RoboDK station: AccelerationCalculation.rdk

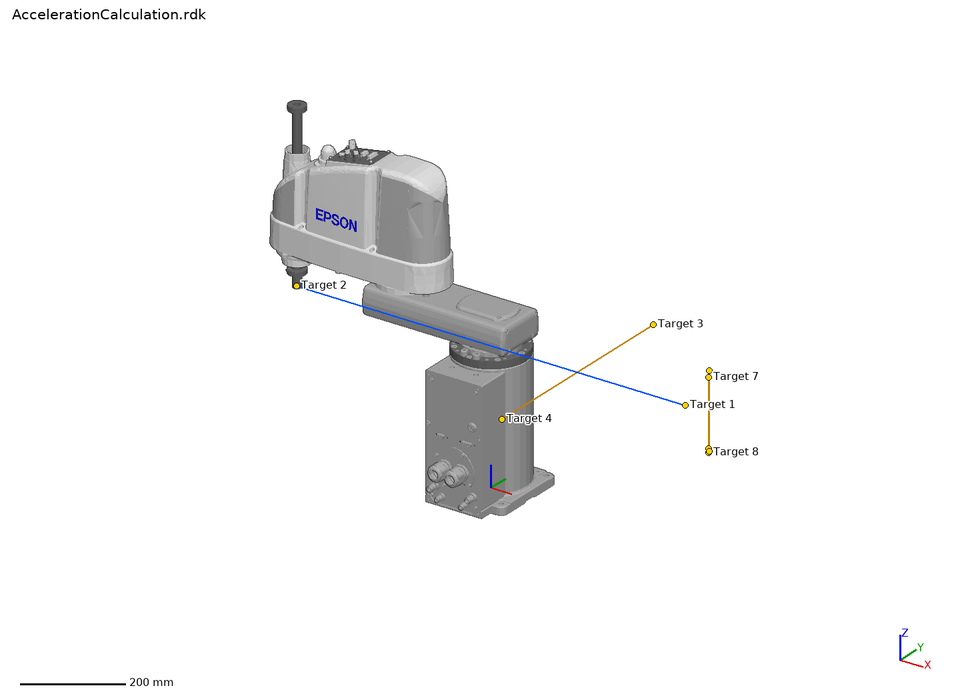
[picture v0: the station drawn from its stored meshes, robots at their saved joint values, targets as dots, program paths as lines]
Station AccelerationCalculation (saved by RoboDK 5.9.6). Poses are relative to the parent item; angles as X-Y-Z fixed-axis rotations.
  - frame Epson_G6_451s Base at (0, 0, 0) mm
    - robot Epson_G6_451s: 4 axes
        modified DH rows (alpha deg, a mm, theta deg, d mm): 0, 0, 0, 0; 0, 200, 0, 0; 0, 250, 0, -180 linear; 180, 0, 0, 0
        joint limits [-62, -142, -180, -360] to [242, 142, 0, 360]; home [0, 0, 0, 0]; saved at [180, 0, 0, 0]
    - target Target 1 (Cartesian target) at (450, 0, 300) mm, rotated rx 180 ry 0 rz 0 deg; joints [0, 0, 0, 0] of Epson_G6_451s
    - target Target 2 (Cartesian target) at (-450, 0, 300) mm, rotated rx 180 ry 0 rz 180 deg; joints [180, 0, 0, 0] of Epson_G6_451s
    - target Target 3 (Cartesian target) at (200, 250, 300) mm, rotated rx 180 ry 0 rz 90 deg; joints [0, 90, 0, 0] of Epson_G6_451s
    - target Target 4 (Cartesian target) at (200, -250, 300) mm, rotated rx 180 ry 0 rz -90 deg; joints [0, -90, 0, 0] of Epson_G6_451s
    - target Target 5 (Cartesian target) at (200, 250, 300) mm, rotated rx 180 ry 0 rz 90 deg; joints [0, 90, 0, 0] of Epson_G6_451s
    - target Target 6 (Cartesian target) at (450, 0, 300) mm, rotated rx 180 ry 0 rz 0 deg; joints [0, 0, 0, 0] of Epson_G6_451s
    - target Target 7 (Cartesian target) at (416.68, 124.7, 300) mm, rotated rx 180 ry 0 rz 29.92 deg; joints [0, 29.92, 0, 0] of Epson_G6_451s
    - target Target 8 (Cartesian target) at (416.68, 124.7, 141) mm, rotated rx 180 ry 0 rz 29.92 deg; joints [0, 29.92, -159, 0] of Epson_G6_451s
    - target Target 9 (Cartesian target) at (416.68, 124.7, 150) mm, rotated rx 180 ry 0 rz 29.92 deg; joints [0, 29.92, -150, 0] of Epson_G6_451s
    - target Target 10 (Cartesian target) at (450, 0, 300) mm, rotated rx 180 ry 0 rz 0 deg; joints [0, 0, 0, 0] of Epson_G6_451s
    - target Target 11 (Cartesian target) at (-450, 0, 300) mm, rotated rx 180 ry 0 rz 180 deg; joints [180, 0, 0, 0] of Epson_G6_451s
    - target Target 12 (Cartesian target) at (400.78, 148.95, 130) mm, rotated rx 180 ry 0 rz 36.57 deg; joints [0, 36.57, -170, 0] of Epson_G6_451s
    - target Target 13 (Cartesian target) at (400.78, 148.95, 300) mm, rotated rx 180 ry 0 rz 36.57 deg; joints [0, 36.57, 0, 0] of Epson_G6_451s
    - target Target 14 (Cartesian target) at (450, 0, 300) mm, rotated rx 180 ry 0 rz -10 deg; joints [0, 0, 0, -350] of Epson_G6_451s
    - target Target 15 (Cartesian target) at (450, 0, 300) mm, rotated rx 180 ry 0 rz 10 deg; joints [0, 0, 0, 350] of Epson_G6_451s
  - program Joint1 (4 instructions, listed below)
  - Python program GetJointData (listed below)
  - program Joint2 (3 instructions, listed below)
  - program Joint3_Power (61 instructions, listed below)
  - program Joint1_Power (51 instructions, listed below)
  - program Joint2_Power (70 instructions, listed below)
  - program Joint3 (4 instructions, listed below)
  - program Prog6 (5 instructions, listed below)
  - Python program SpeedOutput (listed below)
  - Python program FullOutput (listed below)
  - Python program FullOutputCSVJointMove (listed below)
  - Python program FullOutputCSVLinearMove (listed below)
  - Python program Prog9 (listed below)
  - program Prog14 (61 instructions, listed below)
  - program Joint4 (3 instructions, listed below)
  - program Joint4_Power (60 instructions, listed below)
  - program Prog17 (10 instructions, listed below)
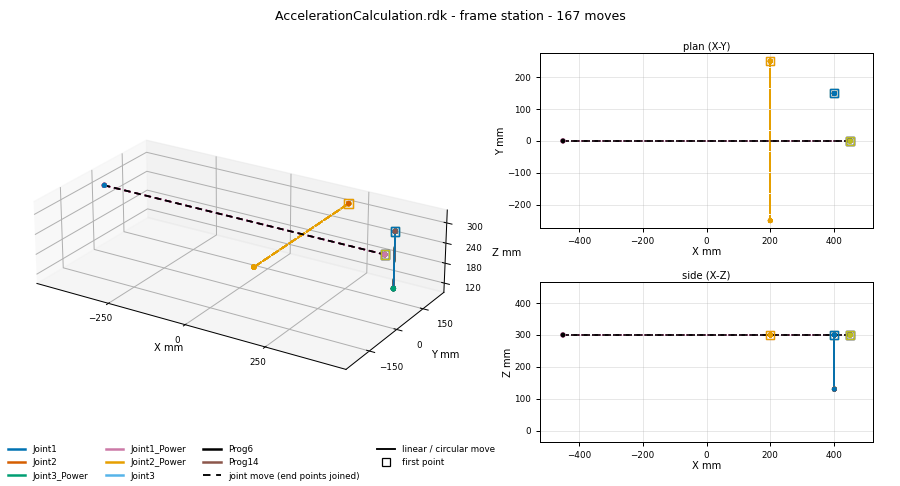
[picture p0: tool path of AccelerationCalculation.rdk in frame station, 167 of 167 moves have a stored position in this frame; points joined in program order, loops and branches not executed]

--- program Joint1 (robot Epson_G6_451s) ---
  Set Ref.: Epson_G6_451s Base
  Set speed (42.0 deg/s)
  MoveJ (Target 1)
  MoveJ (Target 2)

--- Python program GetJointData ---
from robodk import robolink, robomath
import matplotlib.pyplot as plt
from robodk.robolink import *
from robodk.robomath import *
import csv

# Connect to RoboDK
RDK = Robolink()


# Select your program by name
program = RDK.Item('Joint1', robolink.ITEM_TYPE_PROGRAM)  # Change name as needed

# Run the program (optional — comment out if already simulated)
program.RunProgram()

# Retrieve joint data
data_all = program.InstructionListJoints(mm_step=1, deg_step=1, flags=3)
data_all = data_all[1:]

joint_data = data_all[0]
print(joint_data)

# Output file path (can be absolute or relative)
csv_file = 'C:/Users/kytho/Desktop/robot_data.csv'

if program.Valid():
    # Write to CSV

    # Add header row (titles) and append a cumulative Time_Total column
    header = [
        'J1_Position', 'J2_Position', 'J3_Position', 'J4_Position', 'Error',
        'MM_Step', 'Deg_step', 'Move_ID', 'Time', 'Time_Total', 'X', 'Y', 'Z',
        'J1_Velocity', 'J2_Velocity', 'J3_Velocity', 'J4_Velocity',
        'J1_Acceleration', 'J2_Acceleration', 'J3_Acceleration', 'J4_Acceleration'
    ]

    with open(csv_file, "w", newline="") as file:
        writer = csv.writer(file)
        # write header first (move all data one row down)
        writer.writerow(header)

        # compute cumulative Time_Total (Time is expected at index 8)
        time_total = 0.0
        for row in joint_data:
            # keep the original data unchanged; append Time_Total after Time
            new_row = list(row)
            try:
                # read time delta from column index 8
                t_delta = float(row[8])
            except Exception:
                # if parsing fails, treat delta as 0.0
                t_delta = 0.0
            time_total += t_delta
            # insert cumulative time after the existing Time column
            new_row.insert(9, time_total)
            writer.writerow(new_row)

    print("Joint data successfully written to 'robot_data.csv'")
    print("Total Time:",time_total)
else:
    print("No valid program selected.")

--- program Joint2 (robot Epson_G6_451s) ---
  Set Ref.: Epson_G6_451s Base
  MoveJ (Target 5)
  MoveJ (Target 4)

--- program Joint3_Power (robot Epson_G6_451s) ---
  Set Ref.: Epson_G6_451s Base
  Set speed (1182.2 mm/s)
  MoveJ (Target 13)
  MoveL (Target 13)
  MoveL (Target 12)
  Pause 1.0 s
  MoveL (Target 13)
  Pause 1.0 s
  Set speed (1070.0 mm/s)
  MoveL (Target 13)
  MoveL (Target 12)
  Pause 1.0 s
  MoveL (Target 13)
  Pause 1.0 s
  Set speed (953.1 mm/s)
  MoveL (Target 13)
  MoveL (Target 12)
  Pause 1.0 s
  MoveL (Target 13)
  Pause 1.0 s
  Set speed (828.6 mm/s)
  MoveL (Target 13)
  MoveL (Target 12)
  Pause 1.0 s
  MoveL (Target 13)
  Pause 1.0 s
  Set speed (716.0 mm/s)
  MoveL (Target 13)
  MoveL (Target 12)
  Pause 1.0 s
  MoveL (Target 13)
  Pause 1.0 s
  Set speed (595.8 mm/s)
  MoveL (Target 13)
  MoveL (Target 12)
  Pause 1.0 s
  MoveL (Target 13)
  Pause 1.0 s
  Set speed (477.4 mm/s)
  MoveL (Target 13)
  MoveL (Target 12)
  Pause 1.0 s
  MoveL (Target 13)
  Pause 1.0 s
  Set speed (358.1 mm/s)
  MoveL (Target 13)
  MoveL (Target 12)
  Pause 1.0 s
  MoveL (Target 13)
  Pause 1.0 s
  Set speed (238.7 mm/s)
  MoveL (Target 13)
  MoveL (Target 12)
  Pause 1.0 s
  MoveL (Target 13)
  Pause 1.0 s
  Set speed (119.3 mm/s)
  MoveL (Target 13)
  MoveL (Target 12)
  Pause 1.0 s
  MoveL (Target 13)

--- program Joint1_Power (robot Epson_G6_451s) ---
  Set Ref.: Epson_G6_451s Base
  Set speed (420.0 deg/s)
  MoveJ (Target 10)
  MoveJ (Target 11)
  MoveJ (Target 10)
  Pause 1.0 s
  Set speed (378.0 deg/s)
  MoveJ (Target 10)
  MoveJ (Target 11)
  MoveJ (Target 10)
  Pause 1.0 s
  Set speed (336.0 deg/s)
  MoveJ (Target 10)
  MoveJ (Target 11)
  MoveJ (Target 10)
  Pause 1.0 s
  Set speed (294.0 deg/s)
  MoveJ (Target 10)
  MoveJ (Target 11)
  MoveJ (Target 10)
  Pause 1.0 s
  Set speed (251.0 deg/s)
  MoveJ (Target 10)
  MoveJ (Target 11)
  MoveJ (Target 10)
  Pause 1.0 s
  Set speed (210.0 deg/s)
  MoveJ (Target 10)
  MoveJ (Target 11)
  MoveJ (Target 10)
  Pause 1.0 s
  Set speed (168.0 deg/s)
  MoveJ (Target 10)
  MoveJ (Target 11)
  MoveJ (Target 10)
  Pause 1.0 s
  Set speed (126.0 deg/s)
  MoveJ (Target 10)
  MoveJ (Target 11)
  MoveJ (Target 10)
  Pause 1.0 s
  Set speed (84.0 deg/s)
  MoveJ (Target 10)
  MoveJ (Target 11)
  MoveJ (Target 10)
  Pause 1.0 s
  Set speed (42.0 deg/s)
  MoveJ (Target 10)
  MoveJ (Target 11)
  MoveJ (Target 10)
  Pause 1.0 s

--- program Joint2_Power (robot Epson_G6_451s) ---
  Set speed (720.0 deg/s)
  Set Ref.: Epson_G6_451s Base
  MoveJ (Target 5)
  MoveJ (Target 4)
  Pause 1.0 s
  MoveJ (Target 5)
  Pause 1.0 s
  Set speed (648.0 deg/s)
  Set Ref.: Epson_G6_451s Base
  MoveJ (Target 5)
  MoveJ (Target 4)
  Pause 1.0 s
  MoveJ (Target 5)
  Pause 1.0 s
  Set speed (576.0 deg/s)
  Set Ref.: Epson_G6_451s Base
  MoveJ (Target 5)
  MoveJ (Target 4)
  Pause 1.0 s
  MoveJ (Target 5)
  Pause 1.0 s
  Set speed (504.0 deg/s)
  Set Ref.: Epson_G6_451s Base
  MoveJ (Target 5)
  MoveJ (Target 4)
  Pause 1.0 s
  MoveJ (Target 5)
  Pause 1.0 s
  Set speed (432.0 deg/s)
  Set Ref.: Epson_G6_451s Base
  MoveJ (Target 5)
  MoveJ (Target 4)
  Pause 1.0 s
  MoveJ (Target 5)
  Pause 1.0 s
  Set speed (360.0 deg/s)
  Set Ref.: Epson_G6_451s Base
  MoveJ (Target 5)
  MoveJ (Target 4)
  Pause 1.0 s
  MoveJ (Target 5)
  Pause 1.0 s
  Set speed (288.0 deg/s)
  Set Ref.: Epson_G6_451s Base
  MoveJ (Target 5)
  MoveJ (Target 4)
  Pause 1.0 s
  MoveJ (Target 5)
  Pause 1.0 s
  Set speed (216.0 deg/s)
  Set Ref.: Epson_G6_451s Base
  MoveJ (Target 5)
  MoveJ (Target 4)
  Pause 1.0 s
  MoveJ (Target 5)
  Pause 1.0 s
  Set speed (144.0 deg/s)
  Set Ref.: Epson_G6_451s Base
  MoveJ (Target 5)
  MoveJ (Target 4)
  Pause 1.0 s
  MoveJ (Target 5)
  Pause 1.0 s
  Set speed (72.0 deg/s)
  Set Ref.: Epson_G6_451s Base
  MoveJ (Target 5)
  MoveJ (Target 4)
  Pause 1.0 s
  MoveJ (Target 5)
  Pause 1.0 s

--- program Joint3 (robot Epson_G6_451s) ---
  Set Ref.: Epson_G6_451s Base
  Set speed (500.0 mm/s)
  MoveL (Target 13)
  MoveL (Target 12)

--- program Prog6 (robot Epson_G6_451s) ---
  Set Ref.: Epson_G6_451s Base
  Set speed (41.0 deg/s)
  MoveJ (Target 10)
  MoveJ (Target 11)
  MoveJ (Target 10)

--- Python program SpeedOutput ---
# This example shows how to quickly calculate the cycle time of a program
# as a function of the linear and joint speeds
#
# Important notes and tips for accurate cycle time calculation:
# https://robodk.com/doc/en/General.html#CycleTime

# Start the RoboDK API
from robodk.robolink import *  # RoboDK API

RDK = Robolink()

# Ask the user to select a program
program = RDK.ItemUserPick('Joint2', ITEM_TYPE_PROGRAM)

# Retrieve the robot linked to the selected program
robot = program.getLink(ITEM_TYPE_ROBOT)

for speed_joints in range(20, 601, 10):
    # Set the robot speed
    robot.setAcceleration(3516.67)
    robot.setSpeed(500, speed_joints)
    # Update the program and retrieve updated information:
    # https://robodk.com/doc/en/PythonAPI/robodk.html#robodk.robolink.Item.Update
    result = program.Update()
    instructions, time, travel, ok, error = result

    # Print the information
    print("Speed", speed_joints)
    print(time)

--- Python program FullOutput ---
# This example shows how to quickly calculate the cycle time of a program
# as a function of the linear and joint speeds
#
# Important notes and tips for accurate cycle time calculation:
# https://robodk.com/doc/en/General.html#CycleTime

# Start the RoboDK API
from robodk.robolink import *  # RoboDK API

RDK = Robolink()

# Ask the user to select a program
program = RDK.ItemUserPick('Joint2', ITEM_TYPE_PROGRAM)

# Retrieve the robot linked to the selected program
robot = program.getLink(ITEM_TYPE_ROBOT)

for speed_joints in range(20, 601, 10):
    # Set the robot speed
    robot.setAccelerationJoints(3516.67)
    robot.setSpeed(500, speed_joints)
    # Update the program and retrieve updated information:
    # https://robodk.com/doc/en/PythonAPI/robodk.html#robodk.robolink.Item.Update
    result = program.Update()
    instructions, time, travel, ok, error = result

    # Print the information
    print("Speed", speed_joints)
    print(time)

for accel_joints in range(100, 4001, 100):
    # Set the robot speed
    robot.setAccelerationJoints(accel_joints)
    robot.setSpeed(500, 520)
    # Update the program and retrieve updated information:
    # https://robodk.com/doc/en/PythonAPI/robodk.html#robodk.robolink.Item.Update
    result = program.Update()
    instructions, time2, travel, ok, error = result

    # Print the information
    print("Acceleration:", accel_joints)
    print(time2)

--- Python program FullOutputCSVJointMove ---
# This example calculates program cycle time as a function of
# joint speed and joint acceleration and writes results to CSV

from robodk.robolink import *  # RoboDK API
import csv
import os

RDK = Robolink()

# Select program
program = RDK.ItemUserPick('Select a program', ITEM_TYPE_PROGRAM)
if not program.Valid():
    raise Exception("No program selected.")

# Get linked robot
robot = program.getLink(ITEM_TYPE_ROBOT)
if not robot.Valid():
    raise Exception("No robot linked to program.")

results = []

# -----------------------------
# SPEED SWEEP
# -----------------------------
for speed_joints in range(20, 3400, 50):

    robot.setAccelerationJoints(1645.795918)
    robot.setSpeed(500, speed_joints)

    result = program.Update()
    instructions, time_val, travel, ok, error = result

    print("Speed:", speed_joints)
    print("Cycle Time:", time_val)

    results.append([speed_joints, time_val, "", ""])

# -----------------------------
# ACCELERATION SWEEP
# -----------------------------
for accel_joints in range(100, 15100, 100):

    robot.setAccelerationJoints(accel_joints)
    robot.setSpeed(1, 420)

    result = program.Update()
    instructions, time_val, travel, ok, error = result

    print("Acceleration:", accel_joints)
    print("Cycle Time:", time_val)

    results.append(["", "", accel_joints, time_val])

# -----------------------------
# WRITE CSV
# -----------------------------
filename = "robodk_cycle_time_results.csv"

with open(filename, mode='w', newline='') as file:
    writer = csv.writer(file)
    writer.writerow(["joint_speed", "cycle_time", "joint_accel", "cycle_time"])
    writer.writerows(results)

print("\nResults saved to:", os.path.abspath(filename))

--- Python program FullOutputCSVLinearMove ---
# This example calculates program cycle time as a function of
# joint speed and joint acceleration and writes results to CSV

from robodk.robolink import *  # RoboDK API
import csv
import os

RDK = Robolink()

# Select program
program = RDK.ItemUserPick('Select a program', ITEM_TYPE_PROGRAM)
if not program.Valid():
    raise Exception("No program selected.")

# Get linked robot
robot = program.getLink(ITEM_TYPE_ROBOT)
if not robot.Valid():
    raise Exception("No robot linked to program.")

results = []

# -----------------------------
# SPEED SWEEP
# -----------------------------
for speed_joints in range(20, 2001, 20):

    robot.setAcceleration(10100.434747)
    robot.setSpeed(speed_joints, 480)

    result = program.Update()
    instructions, time_val, travel, ok, error = result

    print("Speed:", speed_joints)
    print("Cycle Time:", time_val)

    results.append([speed_joints, time_val, "", ""])

# -----------------------------
# ACCELERATION SWEEP
# -----------------------------
for accel_joints in range(100, 50000, 200):

    robot.setAcceleration(accel_joints)
    robot.setSpeed(1180, 480.037)

    result = program.Update()
    instructions, time_val, travel, ok, error = result

    print("Acceleration:", accel_joints)
    print("Cycle Time:", time_val)

    results.append(["", "", accel_joints, time_val])

# -----------------------------
# WRITE CSV
# -----------------------------
filename = "robodk_cycle_time_results.csv"

with open(filename, mode='w', newline='') as file:
    writer = csv.writer(file)
    writer.writerow(["joint_speed", "cycle_time", "joint_accel", "cycle_time"])
    writer.writerows(results)

print("\nResults saved to:", os.path.abspath(filename))

--- Python program Prog9 ---
from robodk.robolink import Robolink, ITEM_TYPE_PROGRAM
import csv
import re
import statistics
from collections import defaultdict

PROGRAM_NAME = "Joint1_Power"
OUT_CSV = r"C:/Users/kytho/Desktop/robot_data_with_pauses.csv"

def pick_pause_dt(joint_rows, dt_index=8):
    """Use median dt from motion samples for pause sampling."""
    dts = []
    for r in joint_rows:
        try:
            dt = float(r[dt_index])
            if dt > 0:
                dts.append(dt)
        except:
            pass
    return statistics.median(dts) if dts else 0.01

def get_events_from_program_tree(program):
    """
    Build ordered events by reading instruction nodes from the RoboDK tree.
    Requires program.ShowInstructions(True).
    """
    program.ShowInstructions(True)  # key workaround: expose instruction nodes in tree

    children = program.Childs()  # returns items in program order (tree order)
    events = []

    # Matches: "Pause 1.0 s" / "Pause 1s" / "Pause 0.5 s"
    pause_re = re.compile(r"^\s*Pause\s*([0-9]*\.?[0-9]+)\s*s?\s*$", re.IGNORECASE)

    for it in children:
        name = it.Name().strip()

        m = pause_re.match(name)
        if m:
            events.append(("PAUSE", float(m.group(1))))
            continue

        n = name.lower()
        if n.startswith("movej") or n.startswith("movel") or n.startswith("movec"):
            events.append(("MOVE", None))
            continue

        # Ignore "Set speed", messages, etc. (add here if you want them handled)

    return events

def main():
    RDK = Robolink()

    program = RDK.Item(PROGRAM_NAME, ITEM_TYPE_PROGRAM)
    if not program.Valid():
        raise Exception(f"Program not found: {PROGRAM_NAME}")

    # --- motion samples (movement only) ---
    data_all = program.InstructionListJoints(mm_step=1, deg_step=1, flags=3)
    data_all = data_all[1:]  # skip header block if present
    joint_rows = data_all[0]
    if not joint_rows:
        raise Exception("No joint data returned by InstructionListJoints().")

    IDX_MOVE_ID = 7
    IDX_DT = 8

    # Group rows by Move_ID in appearance order
    rows_by_move = defaultdict(list)
    move_ids_in_order = []
    seen = set()
    for row in joint_rows:
        mid = row[IDX_MOVE_ID]
        rows_by_move[mid].append(row)
        if mid not in seen:
            seen.add(mid)
            move_ids_in_order.append(mid)

    # --- parse events from program tree (includes Pause items) ---
    events = get_events_from_program_tree(program)

    move_events = sum(1 for e in events if e[0] == "MOVE")
    pause_events = sum(1 for e in events if e[0] == "PAUSE")
    print("MOVE events found:", move_events)
    print("PAUSE events found:", pause_events)

    if pause_events == 0:
        print("WARNING: No pauses detected from program tree items. Check that pause items exist and are named like 'Pause 1.0 s'.")
    if move_events == 0:
        print("WARNING: No MOVE events detected from program tree items. Check that the program contains MoveJ/MoveL instructions.")

    pause_dt = pick_pause_dt(joint_rows, dt_index=IDX_DT)

    # Output header (same as yours)
    header = [
        "J1_Position", "J2_Position", "J3_Position", "J4_Position", "Error",
        "MM_Step", "Deg_step", "Move_ID", "Time", "Time_Total", "X", "Y", "Z",
        "J1_Velocity", "J2_Velocity", "J3_Velocity", "J4_Velocity",
        "J1_Acceleration", "J2_Acceleration", "J3_Acceleration", "J4_Acceleration"
    ]

    time_total = 0.0
    move_ptr = 0
    last_written = None

    with open(OUT_CSV, "w", newline="") as f:
        w = csv.writer(f)
        w.writerow(header)

        for ev_type, ev_val in events:
            if ev_type == "MOVE":
                if move_ptr >= len(move_ids_in_order):
                    continue

                mid = move_ids_in_order[move_ptr]
                move_ptr += 1

                for row in rows_by_move[mid]:
                    new_row = list(row)
                    try:
                        dt = float(row[IDX_DT])
                    except:
                        dt = 0.0

                    time_total += dt
                    new_row.insert(9, time_total)  # Time_Total after Time column
                    w.writerow(new_row)
                    last_written = new_row

            elif ev_type == "PAUSE":
                pause_s = float(ev_val)
                if last_written is None:
                    continue

                remaining = pause_s
                while remaining > 1e-12:
                    dt = pause_dt if remaining > pause_dt else remaining
                    remaining -= dt

                    pause_row = list(last_written)

                    # "Time" is at index 8, "Time_Total" at index 9 (because we inserted it)
                    pause_row[8] = dt

                    # Zero velocities (cols 13..16) and accelerations (17..20)
                    for i in range(13, 17):
                        pause_row[i] = 0.0
                    for i in range(17, 21):
                        pause_row[i] = 0.0

                    time_total += dt
                    pause_row[9] = time_total
                    w.writerow(pause_row)
                    last_written = pause_row

        # Append any leftover motion blocks if events had fewer MOVE entries than motion blocks
        while move_ptr < len(move_ids_in_order):
            mid = move_ids_in_order[move_ptr]
            move_ptr += 1
            for row in rows_by_move[mid]:
                new_row = list(row)
                try:
                    dt = float(row[IDX_DT])
                except:
                    dt = 0.0
                time_total += dt
                new_row.insert(9, time_total)
                w.writerow(new_row)

    print("Wrote:", OUT_CSV)
    print("Total time (motion + inserted pauses):", time_total)

if __name__ == "__main__":
    main()

--- program Prog14 (robot Epson_G6_451s) ---
  Set Ref.: Epson_G6_451s Base
  Set speed (1100.0 mm/s)
  MoveJ (Target 13)
  MoveL (Target 12)
  Pause 1.0 s
  MoveL (Target 13)
  Pause 1.0 s
  Set speed (990.0 mm/s)
  MoveJ (Target 13)
  MoveL (Target 12)
  Pause 1.0 s
  MoveL (Target 13)
  Pause 1.0 s
  Set speed (880.0 mm/s)
  MoveJ (Target 13)
  MoveL (Target 12)
  Pause 1.0 s
  MoveL (Target 13)
  Pause 1.0 s
  Set speed (770.0 mm/s)
  MoveJ (Target 13)
  MoveL (Target 12)
  Pause 1.0 s
  MoveL (Target 13)
  Pause 1.0 s
  Set speed (660.0 mm/s)
  MoveJ (Target 13)
  MoveL (Target 12)
  Pause 1.0 s
  MoveL (Target 13)
  Pause 1.0 s
  Set speed (550.0 mm/s)
  MoveJ (Target 13)
  MoveL (Target 12)
  Pause 1.0 s
  MoveL (Target 13)
  Pause 1.0 s
  Set speed (440.0 mm/s)
  MoveJ (Target 13)
  MoveL (Target 12)
  Pause 1.0 s
  MoveL (Target 13)
  Pause 1.0 s
  Set speed (330.0 mm/s)
  MoveJ (Target 13)
  MoveL (Target 12)
  Pause 1.0 s
  MoveL (Target 13)
  Pause 1.0 s
  Set speed (220.0 mm/s)
  MoveJ (Target 13)
  MoveL (Target 12)
  Pause 1.0 s
  MoveL (Target 13)
  Pause 1.0 s
  Set speed (110.0 mm/s)
  MoveJ (Target 13)
  MoveL (Target 12)
  Pause 1.0 s
  MoveL (Target 13)
  Pause 1.0 s

--- program Joint4 (robot Epson_G6_451s) ---
  Set Ref.: Epson_G6_451s Base
  MoveJ (Target 14)
  MoveJ (Target 15)

--- program Joint4_Power (robot Epson_G6_451s) ---
  Set Ref.: Epson_G6_451s Base
  Set speed (2400.0 deg/s)
  MoveJ (Target 14)
  MoveJ (Target 15)
  Pause 1.0 s
  MoveJ (Target 14)
  Pause 1.0 s
  Set speed (2160.0 deg/s)
  MoveJ (Target 14)
  MoveJ (Target 15)
  Pause 1.0 s
  MoveJ (Target 14)
  Pause 1.0 s
  Set speed (1920.0 deg/s)
  MoveJ (Target 14)
  MoveJ (Target 15)
  Pause 1.0 s
  MoveJ (Target 14)
  Pause 1.0 s
  Set speed (1680.0 deg/s)
  MoveJ (Target 15)
  Pause 1.0 s
  MoveJ (Target 14)
  Pause 1.0 s
  Set speed (1440.7 deg/s)
  MoveJ (Target 14)
  MoveJ (Target 15)
  Pause 1.0 s
  MoveJ (Target 14)
  Pause 1.0 s
  Set speed (1200.0 deg/s)
  MoveJ (Target 14)
  MoveJ (Target 15)
  Pause 1.0 s
  MoveJ (Target 14)
  Pause 1.0 s
  Set speed (960.0 deg/s)
  MoveJ (Target 14)
  MoveJ (Target 15)
  Pause 1.0 s
  MoveJ (Target 14)
  Pause 1.0 s
  Set speed (720.0 deg/s)
  MoveJ (Target 14)
  MoveJ (Target 15)
  Pause 1.0 s
  MoveJ (Target 14)
  Pause 1.0 s
  Set speed (480.0 deg/s)
  MoveJ (Target 14)
  MoveJ (Target 15)
  Pause 1.0 s
  MoveJ (Target 14)
  Pause 1.0 s
  Set speed (240.0 deg/s)
  MoveJ (Target 14)
  MoveJ (Target 15)
  Pause 1.0 s
  MoveJ (Target 14)
  Pause 1.0 s

--- program Prog17 (robot Epson_G6_451s) ---
  Set Ref.: Epson_G6_451s Base
  Set speed (500.0 mm/s)
  MoveJ (Target 13)
  MoveL (Target 13)
  MoveL (Target 12)
  Pause 1.0 s
  MoveL (Target 13)
  Pause 1.0 s
  MoveJ (Target 13)
  MoveJ (Target 13)
